// TwinCAT 3 PLC project Untitled1
// ProgramVersion: 3.1.4024.0
// libraries:
//   Tc2_MC2, * (Beckhoff Automation GmbH)
//   Tc2_Standard, * (Beckhoff Automation GmbH)
//   Tc2_System, * (Beckhoff Automation GmbH)
//   Tc3_Module, * (Beckhoff Automation GmbH)
//   VisuDialogs, * (System)
// project tree:
//   DUTs/ DUT.TcTLEO
//   / GlobalTextList.TcGTLO, PlcTask.TcTTO, Visualization Manager.TcVMO (not stored)
//   POUs/ CheckStatusVanHetSysteem.TcPOU, MAIN.TcPOU
//   VISUs/ Visualization.TcVIS
// real-time tasks:
//   TASK PlcTask: cycle T#10ms, priority 20, ADS port 350
// motion (NC):
//   TASK NC-Task 1 SAF: cycle T#2ms, priority 4, ADS port 501
//   TASK NC-Task 1 SVB: cycle T#10ms, priority 8, ADS port 511
//   AXIS Axis 1 (id 1)
//     Dynamic: Acceleration=9934.44, Deceleration=9934.44, Jerk=29803.3
//     Velo: RefSearch=66.22962, RefSync=66.22962, SlowManual=331.1481, FastManual=1986.8886, Fast=6622.962, Maximum=6622.96
//     OtherSettings: AllowMotionCmdToSlave=true
//     encoder EncType=8
//       EncPara: ScaleFactorNumerator=60, ScaleFactorDenominator=1048576, MaxCount=#xffffffff
//         SoftEndMinControl: Enable=true, Range=-5
//         SoftEndMaxControl: Enable=true, Range=3000
//     drive DrvType=9
//       DrvPara: MaxCount=#xffffffff, DriveControlDWord=#x00030000
//         Analog: VeloReferenz=7285.2582, VeloScale=1.02400649589962, TorqueSetpointScale=10, ScaleFactorActTorque=0.1
//         TimeComp: TaskDelayCycles=1
//     controller CtrType=1
//       CtrPara: PriorControlFactor=1
//         Observer: BandWidth=20
// I/O:
//   DEVICE Device 1 (EtherCAT), AmsNetId 10.100.5.10.2.1
//     Term 1 (EK1200) [EK1200-5000 EtherCAT Power supply (2A E-Bus)]
//       Term 2 (EL1819) [EL1819 16Ch. Dig. Input 24V, 10µs]
//       Term 3 (EL2809) [EL2809 16Ch. Dig. Output 24V, 0.5A]
//       Term 4 (EL3151) [EL3151 1Ch. Ana. Input 4-20mA]
//       Term 5 (EL4004) [EL4004 4Ch. Ana. Output 0-10V, 12bit]
//       Term 6 (EL9011) [EL9011 End Terminal]
//   DEVICE Device 2 (EtherCAT Automation Protocol), AmsNetId 10.100.5.10.3.1
//   DEVICE Device 4 (EtherCAT), AmsNetId 10.100.5.10.5.1
//     Drive 7 (AX5106-0000-0214) [AX5106-0000-0214 EtherCAT Drive (SoE, 1 Ch.)]
//   DEVICE Device 5 (COM Port)
// variable links:
//   NC-Task 1 SAF/Axes/Axis 1 <-> Device 4 (EtherCAT)/Drive 7 (AX5106-0000-0214)
//     Drive/Inputs/In/nDataIn1 <-> AT/Following distance
//     Drive/Inputs/In/nDataIn3[0] <-> AT/Torque/force feedback value
//     Drive/Inputs/In/nDcOutputTime <-> InfoData/DcOutputShift
//     Drive/Inputs/In/nState1 <-> AT/Drive status word @bit 8
//     Drive/Inputs/In/nState2 <-> AT/Drive status word
//     Drive/Inputs/In/nState4 @bit 1 <-> WcState/InputToggle
//     Drive/Inputs/In/nState4 <-> WcState/WcState
//     Drive/Outputs/Out/nCtrl1 <-> MDT/Master control word @bit 8
//     Drive/Outputs/Out/nDataOut1 <-> MDT/Position command value
//     Drive/Outputs/Out/nDataOut4[0] <-> MDT/Torque/force command value
//     Drive/Outputs/Out/nDataOut5 <-> MDT/High velocity limit value
//     Drive/Outputs/Out/nDataOut6 <-> MDT/Low velocity limit value
//     Enc/Inputs/In/nDataIn1 <-> AT/Position feedback 1 value
//     Enc/Inputs/In/nDcInputTime <-> InfoData/DcInputShift
//     Enc/Inputs/In/nState4 @bit 1 <-> WcState/InputToggle
//     Enc/Inputs/In/nState4 <-> WcState/WcState
//   Untitled1/Untitled1 Instance <-> Device 1 (EtherCAT)/Term 1 (EK1200)/Term 3 (EL2809)
//     PlcTask Outputs/MAIN.CheckXas.OutDeurslot <-> Channel 5/Output
//   Untitled1/Untitled1 Instance <-> NC-Task 1 SAF/Axes/Axis 1
//     PlcTask Inputs/MAIN.CheckXas.DePositieVanDeXas <-> Outputs/ToPlc/ActPos
//     PlcTask Inputs/MAIN.CheckXas.DeTorqueVanDeXas <-> Outputs/ToPlc/ActTorque
//     PlcTask Inputs/MAIN.CheckXas.InputSensor1 <-> Drive/Outputs/Out/nCtrl2
//     PlcTask Inputs/MAIN.CheckXas.XasDrive.NcToPlc <-> Outputs/ToPlc
//     PlcTask Outputs/MAIN.CheckXas.XasDrive.PlcToNc <-> Inputs/FromPlc

CONFIGURATION Untitled1
    RESOURCE PLC ON TwinCAT3
        TASK PlcTask(INTERVAL := T#10ms, PRIORITY := 20);
        PROGRAM MAIN WITH PlcTask : MAIN;
    END_RESOURCE
END_CONFIGURATION

// ---- DUTs/DUT.TcTLEO
{attribute 'qualified_only'}
{attribute 'strict'}
{attribute 'to_string'}
TYPE SysteemStatusMogelijkheiden :
(
	Uit,
	Joggen,
	Locatie,
	Torque,
	PowerOff
);
END_TYPE

// ---- POUs/MAIN.TcPOU
PROGRAM MAIN
VAR
CheckXas:CheckStatusVanHetSysteem;
END_VAR

CheckXas();

END_PROGRAM

// ---- POUs/CheckStatusVanHetSysteem.TcPOU
FUNCTION_BLOCK CheckStatusVanHetSysteem
VAR
	//Defenieren van de Xas en functies om deze te manipuleren
	XasDrive: AXIS_REF;
	XasDrivePower: MC_Power;
	DeTorqueVanDeXas AT %I* : LREAL;
	DePositieVanDeXas AT %I* : LREAL;
	StopDeBoot : MC_Stop;
	VeranderDriveOperationMode : MC_WriteDriveOperationMode;
	OutDeurslot   AT %Q* : BOOL;
	CheckDoneVoorStoppen : BOOL:= FALSE;
	SetPosZero_Home : MC_Home;
	KnopSetPositionZero_Home AT %I* :BOOL ;
	
	//Inputs Vanuit HMI en Variabele voor checken van drive status
	KnopDriveAan2 AT %I* : BOOL;
	KnopDriveUit  AT %I* : BOOL;
	IndicatieDriveIsActief   AT %Q* : BOOL;
	KnopStopKnop AT %I* : BOOL;	
	KnopDoorgaan AT %I* : BOOL;	
	
	//Variabele voor het bepalen van de state van het systeem
	StatusVanDeStateVanHetSysteem : SysteemStatusMogelijkheiden :=SysteemStatusMogelijkheiden.PowerOff;
	StatusVanDeStateVanHetSysteemText: STRING;
	KnopJoggModus AT %I* : BOOL;
	KnopLocatieModus  AT %I* : BOOL;
	KnopTorqueControl AT %I* : BOOL;
	IndicatieStatusIsUit   AT %Q* : BOOL;
	IndicatieStatusIsJoggen   AT %Q* : BOOL;
	IndicatieStatusIsLocatie   AT %Q* : BOOL;
	IndicatieStatusIsTorque   AT %Q* : BOOL;
	
	// variabele voor Jogg state
	XasJoggModusFB : MC_MoveVelocity;
	HetTypeJog : (LinksTraag, LinksSnel, RechtsSnel, RechtsTraag, StilStaan);
	KnopJoggModusLinksTraag AT %I* : BOOL;
	KnopJoggModusLinksSnel AT %I* : BOOL;
	KnopJoggModusRechtsTraag AT %I* : BOOL;
	KnopJoggModusRechtsSnel AT %I* : BOOL;
	
	// Variabele voor Locatie state
	XasLocatieModeFB : MC_MoveAbsolute;
	StatusLocatieStatemachine : (WachtenOpNieuweLocatie, Uitvoeren, Bezig, Klaar,Pauzen);
 	DeIngevoerdeTargetPositie AT %I* : LREAL;
	NogAfTeLeggenAfstand AT %Q* : LREAL;
	KnopLocatieUitvoeren AT %I* : BOOL;
	KlaarMetBewegen : BOOL :=FALSE ;
	
	//Variabele voor Torque control
	StatusTorqueStatemachine : (WachtenOpNieuwDoel, Bezig2, Stop);
	DOTorqueDing : MC_TorqueControl;
	DeIngevoerdeTorqueDoel AT %I* : LREAL;
	KnopHervatTorquecontrol AT %I* : BOOL;	
	
	// hoopelijk gelinkde I/O
	InputSensor1 AT %I* : BOOL;
	OutputSysteemIsActiefDeurslot AT %Q* : BOOL;
	SlotDicht: BOOL :=FALSE ;
	SlotOpen: BOOL :=TRUE ;
END_VAR

CheckStateVanHetSysteem();
	CASE StatusVanDeStateVanHetSysteem OF
		SysteemStatusMogelijkheiden.PowerOff:
			SetPowerLow();
			OutputSysteemIsActiefDeurslot:=SlotOpen;
			IndicatieDriveIsActief:=FALSE;
			IndicatieStatusIsUit:=FALSE;
			IndicatieStatusIsJoggen:=FALSE;
			IndicatieStatusIsLocatie:=FALSE;
			IndicatieStatusIsTorque:=FALSE;

		SysteemStatusMogelijkheiden.Uit:
			IndicatieStatusIsUit:=TRUE;
			IndicatieStatusIsJoggen:=FALSE;
			IndicatieStatusIsLocatie:=FALSE;
			IndicatieStatusIsTorque:=FALSE;
			OutputSysteemIsActiefDeurslot:=SlotDicht;
		SysteemStatusMogelijkheiden.Joggen:
			IndicatieStatusIsUit:=FALSE;
			IndicatieStatusIsJoggen:=TRUE;
			IndicatieStatusIsLocatie:=FALSE;
			IndicatieStatusIsTorque:=FALSE;
		IF KnopDriveAan2 THEN
			DoJogStatemachine();
		END_IF
			OutputSysteemIsActiefDeurslot:=SlotDicht;
		SysteemStatusMogelijkheiden.Locatie:
			NogAfTeLeggenAfstand:= DeIngevoerdeTargetPositie - DePositieVanDeXas;
			IndicatieStatusIsUit:=FALSE;
			IndicatieStatusIsJoggen:=FALSE;
			IndicatieStatusIsLocatie:=TRUE;
			IndicatieStatusIsTorque:=FALSE;
		IF KnopDriveAan2 THEN
			DoLocatieStatemachine();
		END_IF
			OutputSysteemIsActiefDeurslot:=SlotDicht;		
		SysteemStatusMogelijkheiden.Torque:
			NogAfTeLeggenAfstand:= DeIngevoerdeTargetPositie - DePositieVanDeXas;
			IndicatieStatusIsUit:=FALSE;
			IndicatieStatusIsJoggen:=FALSE;
			IndicatieStatusIsLocatie:=FALSE;
			IndicatieStatusIsTorque:=TRUE;
		IF KnopDriveAan2 THEN
			DoTorqueStatemachine();
		END_IF
			OutputSysteemIsActiefDeurslot:=SlotDicht;
	END_CASE

ACTION CheckStateVanHetSysteem:
		StopDeBoot
(	Axis:= XasDrive,
	Execute:=FALSE,
	Deceleration:=0,
	Jerk:=0,
	Done=>,
	Busy=>,
	Active=>,
	CommandAborted=>,
	Error=>,
	ErrorID=>,);

SetPosZero_Home(
	Axis:=XasDrive, 
	Execute:=KnopSetPositionZero_Home, 
	Position:=0, 
	HomingMode:=MC_Direct, 
	BufferMode:= , 
	Options:= , 
	bCalibrationCam:= , 
	Done=> , 
	Busy=> , 
	Active=> , 
	CommandAborted=> , 
	Error=> , 
	ErrorID=> );
	
	
	StatusVanDeStateVanHetSysteemText :=TO_STRING(StatusVanDeStateVanHetSysteem);
	
//Power Inputs
IF KnopDriveAan2 THEN
	IndicatieDriveIsActief:=TRUE;
	SetPowerHighElkeKant();
	OutDeurslot:= TRUE;
	StatusVanDeStateVanHetSysteem:=SysteemStatusMogelijkheiden.Uit;
END_IF

IF NOT KnopDriveAan2 THEN
		StopDeBoot
(	Axis:= XasDrive,
	Execute:=TRUE,
	Deceleration:=0,
	Jerk:=0,
	Done=>CheckDoneVoorStoppen,
	Busy=>,
	Active=>,
	CommandAborted=>,
	Error=>,
	ErrorID=>,);
	
	IF CheckDoneVoorStoppen THEN
	StatusVanDeStateVanHetSysteem:=SysteemStatusMogelijkheiden.PowerOff;
	IndicatieDriveIsActief:= FALSE;
	END_IF
END_IF

//evtueel error checken

IF KnopJoggModus AND NOT KnopLocatieModus AND IndicatieDriveIsActief AND NOT KnopTorqueControl THEN
	StatusVanDeStateVanHetSysteem:=SysteemStatusMogelijkheiden.Joggen;
END_IF

IF NOT KnopJoggModus AND NOT KnopLocatieModus AND IndicatieDriveIsActief AND KnopTorqueControl THEN
	StatusVanDeStateVanHetSysteem:=SysteemStatusMogelijkheiden.Torque;
END_IF

IF NOT KnopJoggModus AND  KnopLocatieModus AND IndicatieDriveIsActief AND NOT KnopTorqueControl THEN
	StatusVanDeStateVanHetSysteem:=SysteemStatusMogelijkheiden.Locatie;
END_IF

IF IndicatieDriveIsActief AND  NOT KnopJoggModus AND NOT KnopLocatieModus AND NOT KnopTorqueControl THEN
	StatusVanDeStateVanHetSysteem:=SysteemStatusMogelijkheiden.Uit;
END_IF
END_ACTION

ACTION DoJogStatemachine:
XasJoggModusFB
	(
    Axis:= XasDrive,
	Direction:= 1,
	Velocity :=0 ,
	Execute:=FALSE,
	Deceleration:=0,
	Acceleration :=0,
	Jerk:= ,
	BufferMode:= ,
	Options := ,
	InVelocity => ,
	Active => ,
	Busy => ,
	CommandAborted => ,
	Error => ,
	ErrorID => ,
	);
	
	
CASE HetTypeJog OF
	StilStaan:
XasJoggModusFB
(
	Axis:= XasDrive,
	Direction:= 1,
	Velocity :=0 ,
	Execute:=TRUE,
	Deceleration:=0,
	Acceleration :=0,
	Jerk:= ,
	BufferMode:= ,
	Options := ,
	InVelocity => ,
	Active => ,
	Busy => ,
	CommandAborted => ,
	Error => ,
	ErrorID => ,
	);
	IF KnopJoggModusLinksTraag THEN
		HetTypeJog:=LinksTraag;
	END_IF
	IF KnopJoggModusLinksSnel THEN
		HetTypeJog:=LinksSnel;
	END_IF
	IF KnopJoggModusRechtsTraag THEN
		HetTypeJog:=RechtsTraag;
	END_IF
	IF KnopJoggModusRechtsSnel THEN
		HetTypeJog:=RechtsSnel;
	END_IF

		LinksTraag:
XasJoggModusFB
(
    Axis:= XasDrive,
	Direction:= MC_Positive_Direction ,
	Velocity :=250 ,
	Execute:=TRUE,
	Deceleration:=0,
	Acceleration :=0,
	Jerk:= ,
	BufferMode:= ,
	Options := ,
	InVelocity => ,
	Active => ,
	Busy => ,
	CommandAborted => ,
	Error => ,
	ErrorID => ,
	);
	IF NOT KnopJoggModusLinksTraag THEN
		HetTypeJog:=StilStaan;
	END_IF

		LinksSnel:
XasJoggModusFB
(
    Axis:= XasDrive,
	Direction:= MC_Positive_Direction ,
	Velocity :=500 ,
	Execute:=TRUE,
	Deceleration:=0,
	Acceleration :=0,
	Jerk:= ,
	BufferMode:= ,
	Options := ,
	InVelocity => ,
	Active => ,
	Busy => ,
	CommandAborted => ,
	Error => ,
	ErrorID => ,
	);
	IF NOT  KnopJoggModusLinksSnel THEN
		HetTypeJog:=StilStaan;
	END_IF

		RechtsSnel:
XasJoggModusFB
(
    Axis:= XasDrive,
	Direction:= MC_Negative_Direction,
	Velocity :=500 ,
	Execute:=TRUE,
	Deceleration:=0,
	Acceleration :=0,
	Jerk:= ,
	BufferMode:= ,
	Options := ,
	InVelocity => ,
	Active => ,
	Busy => ,
	CommandAborted => ,
	Error => ,
	ErrorID => ,
	);
	IF NOT KnopJoggModusRechtsSnel THEN
		HetTypeJog:=StilStaan;
	END_IF

	
	RechtsTraag:
XasJoggModusFB
(
    Axis:= XasDrive,
	Direction:= MC_Negative_Direction,
	Velocity :=250,
	Execute:=TRUE,
	Deceleration:=0,
	Acceleration :=0,
	Jerk:= ,
	BufferMode:= ,
	Options := ,
	InVelocity => ,
	Active => ,
	Busy => ,
	CommandAborted => ,
	Error => ,
	ErrorID => ,
	);
	IF NOT KnopJoggModusRechtsTraag THEN
		HetTypeJog:=StilStaan;
	END_IF

END_CASE
END_ACTION

ACTION DoLocatieStatemachine:

		XasLocatieModeFB
(   Axis:= XasDrive,
	Execute:=FALSE,
	Position := 0,
	Velocity :=0 ,
	Deceleration:=0,
	Acceleration :=0,
	Jerk:= ,
	BufferMode:= ,
	Options := ,
	Done => KlaarMetBewegen,
	Active => ,
	Busy => ,
	CommandAborted => ,
	Error => ,
	ErrorID => , );
		StopDeBoot
(	Axis:= XasDrive,
	Execute:=FALSE,
	Deceleration:=0,
	Jerk:=0,
	Done=>,
	Busy=>,
	Active=>,
	CommandAborted=>,
	Error=>,
	ErrorID=>,);
IF KnopStopKnop THEN
	StatusLocatieStatemachine := Pauzen;
END_IF

CASE StatusLocatieStatemachine OF 
	WachtenOpNieuweLocatie:
	IF KnopLocatieUitvoeren THEN
		StatusLocatieStatemachine:= Uitvoeren;
	END_IF
	Uitvoeren:
	XasLocatieModeFB
(	Axis:= XasDrive,
	Execute:=TRUE,
	Position := DeIngevoerdeTargetPositie,
	Velocity :=500 ,
	Deceleration:=0,
	Acceleration :=0,
	Jerk:= ,
	BufferMode:= ,
	Options := ,
	Done => KlaarMetBewegen,
	Active => ,
	Busy => ,
	CommandAborted => ,
	Error => ,
	ErrorID => , );
	StatusLocatieStatemachine:= Bezig;
	
	Bezig:
	IF KlaarMetBewegen THEN
		StatusLocatieStatemachine:= Klaar;
	END_IF
	Klaar:
		KlaarMetBewegen:=FALSE;
		XasLocatieModeFB
(   Axis:= XasDrive,
	Execute:=FALSE,
	Position := DeIngevoerdeTargetPositie,
	Velocity :=500 ,
	Deceleration:=0,
	Acceleration :=0,
	Jerk:= ,
	BufferMode:= ,
	Options := ,
	Done => KlaarMetBewegen,
	Active => ,
	Busy => ,
	CommandAborted => ,
	Error => ,
	ErrorID => , );
	StatusLocatieStatemachine:= WachtenOpNieuweLocatie;	
		
	Pauzen:
	StopDeBoot
(	Axis:= XasDrive,
	Execute:=TRUE,
	Deceleration:=0,
	Jerk:=0,
	Done=>,
	Busy=>,
	Active=>,
	CommandAborted=>,
	Error=>,
	ErrorID=>,);
	IF KnopDoorgaan THEN
		StatusLocatieStatemachine:= WachtenOpNieuweLocatie;	
	END_IF


END_CASE
END_ACTION

ACTION DoTorqueStatemachine:

END_ACTION

ACTION SetPowerHighElkeKant:
	XasDrivePower
	(
    Axis:= XasDrive,
    Enable:= TRUE,
    Enable_Positive:= TRUE,
    Enable_Negative:= TRUE,
    Override:= 100,
    BufferMode:= ,
    Options:= ,
    Status=> ,
    Busy=> ,
    Active=> ,
    Error=> ,
    ErrorID=> 
	);
END_ACTION

ACTION SetPowerLow:
	XasDrivePower
	(
    Axis:= XasDrive,
    Enable:= FALSE,
    Enable_Positive:= FALSE,
    Enable_Negative:= FALSE,
    Override:= 100,
    BufferMode:= ,
    Options:= ,
    Status=> ,
    Busy=> ,
    Active=> ,
    Error=> ,
    ErrorID=> 
	);
END_ACTION

END_FUNCTION_BLOCK

// ---- GlobalTextList.TcGTLO
TEXTLIST GlobalTextList
  173 = '%2.5f mm'
  49 = 'Af te leggen afstand: %2.0f'
  589 = 'Af te leggen afstand: %f'
  982 = 'De Locatie van de as: %2.0f'
  448 = 'De Locatie van de as: %2.4f'
  607 = 'De Locatie van de as: %f'
  213 = 'De Status Van het systeem ='
  734 = 'De Status Van het systeem = %s'
  462 = 'De Status Van het systeem =%s'
  651 = 'De Torque van de as: %2.0f'
  380 = 'Drive Aan'
  490 = 'Drive Uit'
  828 = 'Ga naar locatie'
  198 = 'Hervatten'
  67 = 'Jog Modus'
  746 = 'Joggen'
  41 = 'Links Snel'
  634 = 'Links Traag'
  883 = 'Locatie'
  670 = 'Locatie Modus'
  792 = 'Nieuwe invoer'
  691 = 'Rechts Snel'
  999 = 'Rechts Traag'
  264 = 'Status Jog modus'
  837 = 'Status Locatie modus'
  995 = 'Stop'
  9 = 'Systeem Geen modus geselecteerd'
  700 = 'Systeem uit'
  23 = 'Torque control'
  118 = 'Torque control Mode'
END_TEXTLIST

// ---- VISUs/Visualization.TcVIS
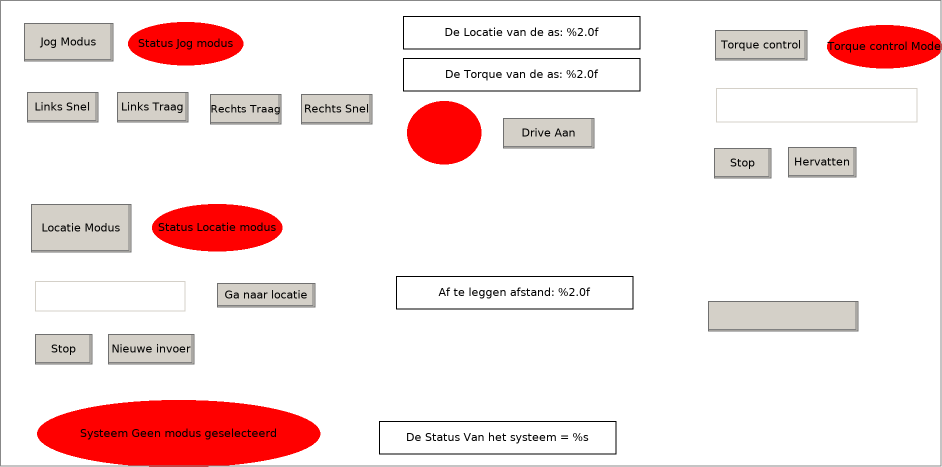
VISUALIZATION Visualization  // 942x467
    Button (503,118 91x30), "Drive Aan"
        toggle MAIN.CheckXas.KnopDriveAan2
    Ellipse (407,101 74x63), colour toggle: MAIN.CheckXas.IndicatieDriveIsActief
    Ellipse (128,22 115x43), "Status Jog modus", colour toggle: MAIN.CheckXas.IndicatieStatusIsJoggen
    Button (27,92 71x30), "Links Snel"
        tap MAIN.CheckXas.KnopJoggModusLinksSnel
    Button (117,92 71x30), "Links Traag"
        tap MAIN.CheckXas.KnopJoggModusLinksTraag
    Button (301,94 71x30), "Rechts Snel"
        tap MAIN.CheckXas.KnopJoggModusRechtsSnel
    Button (210,94 71x30), "Rechts Traag"
        tap MAIN.CheckXas.KnopJoggModusRechtsTraag
    Rectangle (403,16 237x33), "De Locatie van de as: %2.0f", text variable: MAIN.CheckXas.DePositieVanDeXas
    Textfield (35,281 150x30)
        OnMouseClick: write MAIN.CheckXas.DeIngevoerdeTargetPositie via VisuDialogs.Numpad
    Ellipse (152,204 130x47), "Status Locatie modus", colour toggle: MAIN.CheckXas.IndicatieStatusIsLocatie
    Button (217,283 98x24), "Ga naar locatie"
        tap MAIN.CheckXas.KnopLocatieUitvoeren
    Button (24,23 89x38), "Jog Modus"
        toggle MAIN.CheckXas.KnopJoggModus
    Button (31,204 100x48), "Locatie Modus"
        toggle MAIN.CheckXas.KnopLocatieModus
    Ellipse (37,400 283x67), "Systeem Geen modus geselecteerd", colour toggle: MAIN.CheckXas.IndicatieStatusIsUit
    Rectangle (396,276 237x33), "Af te leggen afstand: %2.0f", text variable: MAIN.CheckXas.NogAfTeLeggenAfstand
    Button (35,334 57x30), "Stop"
        tap MAIN.CheckXas.KnopStopKnop
    Button (108,334 86x30), "Nieuwe invoer"
        tap MAIN.CheckXas.KnopDoorgaan
    Button (715,30 92x30), "Torque control"
        toggle MAIN.CheckXas.KnopTorqueControl
    Ellipse (827,25 115x43), "Torque control Mode", colour toggle: MAIN.CheckXas.IndicatieStatusIsTorque
    Button (788,147 68x30), "Hervatten"
        tap MAIN.CheckXas.KnopHervatTorquecontrol
    Button (714,148 57x30), "Stop"
        tap MAIN.CheckXas.KnopStopKnop
    Textfield (716,88 201x34)
        OnMouseClick: write MAIN.CheckXas.DeIngevoerdeTorqueDoel via VisuDialogs.Numpad
    Button (708,301 150x30)
        tap MAIN.CheckXas.KnopSetPositionZero_Home
    Rectangle (403,58 237x33), "De Torque van de as: %2.0f", text variable: MAIN.CheckXas.DeTorqueVanDeXas
    Rectangle (379,421 237x33), "De Status Van het systeem = %s", text variable: MAIN.CheckXas.StatusVanDeStateVanHetSysteemText
END_VISUALIZATION
